FUNCTION_BLOCK FB_5_TransferirBase_SFC
VAR_INPUT
	
	//  SFC-Flags
	SFCPause: BOOL;
	SFCReset: BOOL;

	// Indicadores de sincronización
	Ack: BOOL := TRUE;
	Execute: BOOL;
	
	// Entradas
	PalePresencia: BOOL;
	TpoCintaFuera: TIME;
	TpoRetenedorBaja: TIME;
	
END_VAR
VAR_OUTPUT
	
	// Indicadores de sincronización
	Ready: BOOL;	
	Done: BOOL;
	
	// Salidas
	CintaMotorActiva: BOOL;
	CintaRetenedorBaja: BOOL;
	CintaSeparadorSube: BOOL;
	
END_VAR
VAR
END_VAR

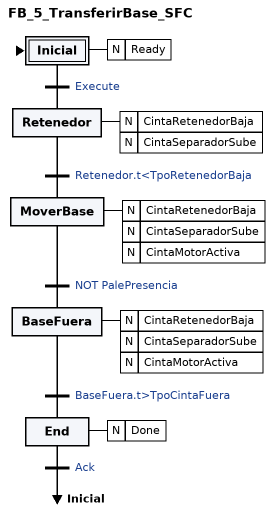
INITIAL_STEP Inicial:
    Ready(N);
END_STEP
TRANSITION FROM Inicial TO Retenedor
    := Execute;
END_TRANSITION
STEP Retenedor:
    CintaRetenedorBaja(N);
    CintaSeparadorSube(N);
END_STEP
TRANSITION FROM Retenedor TO MoverBase
    := Retenedor.t<TpoRetenedorBaja;
END_TRANSITION
STEP MoverBase:
    CintaRetenedorBaja(N);
    CintaSeparadorSube(N);
    CintaMotorActiva(N);
END_STEP
TRANSITION FROM MoverBase TO BaseFuera
    := NOT PalePresencia;
END_TRANSITION
STEP BaseFuera:
    CintaRetenedorBaja(N);
    CintaSeparadorSube(N);
    CintaMotorActiva(N);
END_STEP
TRANSITION FROM BaseFuera TO End
    := BaseFuera.t>TpoCintaFuera;
END_TRANSITION
STEP End:
    Done(N);
END_STEP
TRANSITION FROM End TO Inicial
    := Ack;
END_TRANSITION

END_FUNCTION_BLOCK

(* stored: Version 1.1.0.1, ProductVersion 3.1.4024.12
   POU FB_5_TransferirBase_SFC: Id {83633804-3e25-4538-b573-47cee656cfba}, SpecialFunc None *)
